Fanuc KAREL source: NC0047.KL

-- PROVISIONAL review KL for V940-1; original PC SHA256 93717fba10466c7931d201a2f16a6c9c357c4500172de3b7401d9007e1c01e61
-- Incomplete behavior may be omitted. Consult companion uncertainty JSON. Do not deploy.
PROGRAM NC0047
%NOLOCKGROUP
-- UNRESOLVED_LOCAL_POOL 1 cells at code offset 3; source declarations unknown
-- DIRECT_LOCAL_WORD_ACCESS alone does not prove INTEGER, REAL, or BOOLEAN
BEGIN
  -- V9_CONDITION_STACK_HINT 5 bounded expression windows; static native code-base-relative target link; source arms held
  -- UNRESOLVED_PC offsets 0-8; opcodes 2B,2C,7B
  -- UNRESOLVED_PC offsets 13-20; opcodes 9D,23
  -- UNRESOLVED_PC offsets 25-38; opcodes 21,9D,57,79
  -- UNRESOLVED_PC offsets 43-60; opcodes 21,40,41,42
  -- UNRESOLVED_PC offsets 65-78; opcodes 21,9D,57,79
  -- UNRESOLVED_PC offsets 83-100; opcodes 21,40,41,42
  -- UNRESOLVED_PC offsets 105-118; opcodes 21,9D,57,79
  -- UNRESOLVED_PC offsets 123-140; opcodes 21,40,41,42
  -- UNRESOLVED_PC offsets 145-158; opcodes 21,9D,57,79
  -- UNRESOLVED_PC offsets 163-180; opcodes 21,40,41,42
  -- UNRESOLVED_PC offsets 185-198; opcodes 21,9D,57,79
  -- UNRESOLVED_PC offsets 203-220; opcodes 21,40,41,42
  -- UNRESOLVED_PC offsets 225-255; opcodes 21,9D,52,23,7A,40,41,42
  -- UNRESOLVED_PC offsets 260-284; opcodes 21,2E,52,23,7A,43
  -- UNRESOLVED_PC offsets 289-307; opcodes 21,2E,52,23
  -- UNRESOLVED_PC offsets 317-322; opcodes 7A
  -- UNRESOLVED_PC offsets 327-345; opcodes 21,2E,52,23
  -- UNRESOLVED_PC offsets 350-366; opcodes 7A,40,41,42
  -- UNRESOLVED_PC offsets 371-395; opcodes 21,2E,52,23,7A,43
  -- UNRESOLVED_PC offsets 400-418; opcodes 21,2E,52,23
  -- UNRESOLVED_PC offsets 428-433; opcodes 7A
  -- UNRESOLVED_PC offsets 438-456; opcodes 21,2E,52,23
  -- UNRESOLVED_PC offsets 461-477; opcodes 7A,40,41,42
  -- UNRESOLVED_PC offsets 482-506; opcodes 21,2E,52,23,7A,43
  -- UNRESOLVED_PC offsets 511-529; opcodes 21,2E,52,23
  -- UNRESOLVED_PC offsets 539-544; opcodes 7A
  -- UNRESOLVED_PC offsets 549-567; opcodes 21,2E,52,23
  -- UNRESOLVED_PC offsets 572-588; opcodes 7A,40,41,42
  -- UNRESOLVED_PC offsets 593-617; opcodes 21,2E,52,23,7A,43
  -- UNRESOLVED_PC offsets 622-640; opcodes 21,2E,52,23
  -- UNRESOLVED_PC offsets 650-655; opcodes 7A
  -- UNRESOLVED_PC offsets 660-678; opcodes 21,2E,52,23
  -- UNRESOLVED_PC offsets 683-699; opcodes 7A,40,41,42
  -- UNRESOLVED_PC offsets 704-728; opcodes 21,2E,52,23,7A,43
  -- UNRESOLVED_PC offsets 733-751; opcodes 21,2E,52,23
  -- UNRESOLVED_PC offsets 761-766; opcodes 7A
  -- UNRESOLVED_PC offsets 771-789; opcodes 21,2E,52,23
  -- UNRESOLVED_PC offsets 799-803; opcodes 7F
  -- UNRESOLVED_PC offsets 808-812; opcodes 27,AA
  -- UNRESOLVED_PC offsets 817-821; opcodes 7F
END NC0047
